Staubli VAL3: stop.pgx

public program stop()
begin
    //\brief
  //
  //\Issue
  //22: call user event program
  //
//!Issue 22: call user event program
  call prg:onSystemStop()
  call rob:stop()
  call ui:stop()
  call msl:stop()
  call cleanUpDataBase()
  resetMotion()
  //
  cls()
  title(sCopyRight+sVersion)
  gotoxy(3,6)
  put("Press RUN to restart application")
  bStartUp=false
end
